// TwinCAT 3 PLC project PLC_OCR
// ProgramVersion: 3.1.4024.0
// libraries:
//   Tc2_Standard, * (Beckhoff Automation GmbH)
//   Tc2_System, * (Beckhoff Automation GmbH)
//   Tc3_Module, * (Beckhoff Automation GmbH)
//   Tc3_Vision, * (Beckhoff Automation GmbH)
// project tree:
//   / PlcTask.TcTTO
//   POUs/ F_GetROI.TcPOU, MAIN.TcPOU
// real-time tasks:
//   TASK PlcTask: cycle T#20ms, priority 20, ADS port 350
//   TASK VnTask ImgAcq (FileSource1): cycle T#10ms, priority 5, ADS port 351

CONFIGURATION PLC_OCR
    RESOURCE PLC ON TwinCAT3
        TASK PlcTask(INTERVAL := T#20ms, PRIORITY := 20);
        PROGRAM MAIN WITH PlcTask : MAIN;
    END_RESOURCE
END_CONFIGURATION

// ---- POUs/MAIN.TcPOU
PROGRAM MAIN
VAR
	bInitialized 		: 	BOOL := FALSE;
	bDeinitialize		:	BOOL;
	bCheck				:	BOOL;
	fbInit 				: 	FB_VN_InitializeFunction;	
	nReturnCode			:   UDINT;
	
	hr					:	HRESULT;
	hrCheck				:	HRESULT;
	hrDeinitialize		:	HRESULT;
	hrOCR				:	HRESULT;
	fbCameraControl		:	FB_VN_FileSourceControl;
	eCameraState		:	ETcVnCameraState;
	sFileName 			: 	STRING;
	ImageCounter		:	UINT;

	stPixelFormat		:	TcVnPixelFormat;
	stRoi				:	TcVnRectangle_UDINT;
	fThreshold			:	LREAL;
	bInvertImage		:	BOOL := TRUE;
	
	ipOriginalImage		:	ITcVnImage; 
	ipBinaryImage		:	ITcVnImage; 
	ipThreshBorder		:	ITcVnImage;
	ipStructElem		: 	ITcvnImage;
	ipOriginImageDisp	:	ITcVnDisplayableImage;
	ipBinImageDisp		:	ITcVnDisplayableImage;
	ipThreshBorderDisp	:	ITcVnDisplayableImage;
	
	aRedColor			: 	TcVnVector4_LREAL := [255,0,0];
	aGreenColor			: 	TcVnVector4_LREAL := [0,255,0];
	aBlueColor			: 	TcVnVector4_LREAL := [0,0,255];
	aWhiteColor			: 	TcVnVector4_LREAL := [255,255,255];
	
	// OCR
	bUseExpFunction		:	BOOL := FALSE;
	ipOCRResult 		:	ITcVnContainer; (* Returns the detected characters (ContainerType_Vector_String_SINT) *)
	sText 				: 	STRING(255);
	nStringLenght		:	INT;

	// OCR Exp
	sPattern			:	STRING;			(* String template containing the format in which characters are presented *)
	eOcrOptions			:	UDINT;			(* Specifies which options must be applied to the function (ETcVnOcrOptions) *)
	ipBoundingBoxes		:	ITcVnContainer;	(* Returns the corresponding bounding boxes of the detected characters (ContainerType_Vector_TcVnRectangle_DINT, optional, set to 0 if not required) *)
	ipConfidences		:	ITcVnContainer;	(* Returns the corresponding classification confidences of the detected characters (ContainerType_Vector_REAL, optional, set to 0 if not required) *)
	fMinConfidence		:	REAL;			(* Returns the minimum value of the confidences *)
	
	nNumberOfElements	: 	ULINT;
	nIterator			: 	ULINT;
	aConfidences		:	ARRAY [0..11] OF REAL;
	stRectangle			:	TcVnRectangle_DINT;
END_VAR

// Disclaimer

// This publication contains statements about the suitability of our products for certain
// areas of application. These statements are based on typical features of our products.
// The examples shown in this publication are for demonstration purposes only.
// The information provided herein should not be regarded as specific operation characteristics.
// It is incumbent on the customer to check and decide whether a product is suitable for use
// in a particular application. We do not give any warranty that the source code which is
// made available with this publication is complete or accurate.

// THE SAMPLE CODE CONTAINED IN THIS PUBLICATION IS PROVIDED “AS IS” WITHOUT WARRANTY OF ANY KIND,
// EITHER EXPRESSED, IMPLIED OR STATUTORY, INCLUDING WITHOUT LIMITATION, ANY WARRANTY WITH RESPECT TO NON-INFRINGEMENT,
// FREEDOM FROM PROPRIETARY RIGHTS OF THIRD PARTIES OR FITNESS FOR ANY PARTICULAR PURPOSE.

// This publication may be changed from time to time without prior notice.
// No liability is assumed for errors and/or omissions.
// Our products are described in detail in our data sheets and documentations.
// Product-specific warnings and cautions must be observed.
// For the latest version of our data sheets and documentations visit our website (www.beckhoff.de).

// © Beckhoff Automation GmbH & Co. KG, December 2023

// The reproduction, distribution and utilization of this document as well as the communication
// of its contents to others without express authorization is prohibited. 
// Offenders will be held liable for the payment of damages.
// All rights reserved in the event of the grant of a patent, utility model or design.

//	==========================================================================================

// SAMPLE - OCR (Optical Character Recognition)
//	-------------------------------------------------------

// Steps To Do:
// ------------
// 1. Add the sample images to the FileSource1 Control
// 2. Activate the Configuration -> Start TwinCAT System and PLC to run -> watch the results in the ADS Image Watch
// 3. Switch between OCR standard and expert function with bUseExpFunction

// Load OCR Model
IF NOT bInitialized THEN
	fbInit(eFunction := TCVN_IF_OCR, nOptions := ETcVnOcrModelType.TCVN_OMT_NUMBERS_SC_UCLETTERS OR ETcVnOcrModelType.TCVN_OMT_NUMBERS_SC OR ETcVnOcrModelType.TCVN_OMT_UCLETTERS, bStart := TRUE);
	
	IF NOT fbInit.bBusy THEN
		fbInit(bStart := FALSE);
		IF NOT fbInit.bError THEN
			bInitialized := TRUE;
			nReturnCode := fbInit.nErrorId AND 16#FFF;
		ELSE
			nReturnCode := fbInit.nErrorId AND 16#FFF;
		END_IF
	END_IF
END_IF

// Check if Model is initialized
IF bCheck THEN
	bCheck := FALSE;
	hrCheck := F_VN_CheckFunctionInitialization(eFunction := TCVN_IF_OCR, nOptions := ETcVnOcrModelType.TCVN_OMT_NUMBERS_SC, hrPrev := S_OK);
END_IF

// Unload OCR Model
IF bDeinitialize THEN
	bDeinitialize := FALSE;
	hrDeinitialize := F_VN_DeinitializeFunction(eFunction:= TCVN_IF_OCR, nOptions:= ETcVnOcrModelType.TCVN_OMT_NUMBERS_SC, hrPrev:= S_OK);
	bInitialized := FALSE;
END_IF

// Get Camera State
eCameraState := fbCameraControl.GetState();
	
// CameraControl is in error state, so try to reset the camera connection
IF eCameraState = TCVN_CS_ERROR THEN
	hr := fbCameraControl.Reset();

// Camera not yet streaming
ELSIF eCameraState < TCVN_CS_ACQUIRING THEN
	hr := fbCameraControl.StartAcquisition();

// Camera streaming
ELSIF eCameraState = TCVN_CS_ACQUIRING THEN	
	
	hr := fbCameraControl.GetCurrentImageAndFileName(ipImage := ipOriginalImage, sFileName := sFileName, 80);
	
	IF bInitialized AND SUCCEEDED(hr) AND ipOriginalImage <> 0 THEN
		
		ImageCounter := ImageCounter + 1;
		
		// Check pixel format and prepare work image
		hr := F_VN_GetPixelFormat(ipOriginalImage, stPixelFormat, hr);			
		IF stPixelFormat.nChannels = 3 AND stPixelFormat.ePixelEncoding = TCVN_PE_NONE THEN
			hr := F_VN_ConvertColorSpace(ipOriginalImage, ipBinaryImage, TCVN_CST_RGB_TO_GRAY, hr);			
		ELSE
			hr := F_VN_CopyImage(ipOriginalImage, ipBinaryImage, hr);
		END_IF
		
		// Helper funtion to get ROI and threshold value according to sample image
		F_GetROI(sFileName, stRoi, fThreshold, bInvertImage, sPattern);
			 
		// Set ROI and draw rectangle
		hr := F_VN_SetRoi_TcVnRectangle_UDINT(stRoi, ipBinaryImage, hr);
		hr := F_VN_DrawRectangle_TcVnRectangle_UDINT(stRoi, ipOriginalImage, aRedColor, 2, hr);
		
		// Filter Image 
		// Add or replace pre-processing functions if needed
		hr := F_VN_CreateStructuringElement(ipStructElem, ETcVnStructuringElementShape.TCVN_SES_RECTANGLE, 3,3, hr);
		hr := F_VN_MorphologicalOperator(ipBinaryImage, ipBinaryImage, ETcvnMorphologicalOperator.TCVN_MO_OPENING, ipStructElem, hr);	
		
		// Invert image depending on bright or dark text color 
		IF bInvertImage THEN
			hr := F_VN_Threshold(ipBinaryImage, ipBinaryImage, fThreshold, 255, TCVN_TT_BINARY_INV, hr);
		ELSE
			hr := F_VN_Threshold(ipBinaryImage, ipBinaryImage, fThreshold, 255, TCVN_TT_BINARY, hr);
		END_IF
		
		// Remove border objects
		hr := F_VN_BrightBorderObjects(ipBinaryImage, ipThreshBorder, hr);
		hr := F_VN_SubtractImages(ipBinaryImage, ipThreshBorder, ipBinaryImage, hr);
	
		// Read characters
		IF NOT bUseExpFunction THEN
			hrOCR := F_VN_OCR(
					ipSrcImage		:= ipBinaryImage,
					eModel			:= ETcVnOcrModelType.TCVN_OMT_NUMBERS_SC_UCLETTERS,
					ipCharacters	:= ipOCRResult,
					hrPrev			:= hr);
		ELSE
			hrOCR := F_VN_OCRExp(
					ipSrcImage		:= ipBinaryImage,
					eModel			:= ETcVnOcrModelType.TCVN_OMT_NUMBERS_SC or ETcVnOcrModelType.TCVN_OMT_UCLETTERS,
					ipCharacters	:= ipOCRResult, 
					sPattern		:= sPattern,
					eOcrOptions		:= eOcrOptions,
					ipBoundingBoxes	:= ipBoundingBoxes, 
					ipConfidences	:= ipConfidences,
					hrPrev			:= hr,
					fMinConfidence	=> fMinConfidence);
		END_IF
				
		// Check if characters were found
		hr := F_VN_GetNumberOfElements(ipOCRResult, nNumberOfElements, hrOCR);
		IF SUCCEEDED(hr) AND nNumberOfElements > 0 THEN
			// Export character to string
			hr := F_VN_ExportSubContainer_String(ipOCRResult, 0, sText, 255, hr);
			nStringLenght := LEN(sText);
			
			// Write text result to filtered and original image
			hr := F_VN_PutText(sText, ipBinaryImage, 12, 12, TCVN_FT_HERSHEY_PLAIN, 1, aWhiteColor, hr);
			hr := F_VN_PutText(sText, ipOriginalImage, stRoi.nX + 5, stRoi.nY + 25, TCVN_FT_HERSHEY_DUPLEX, 1, aGreenColor, hr);
			
			IF bUseExpFunction THEN 
				// Get number of Confidence elements and export them if array is large enough 
				MEMSET(ADR(aConfidences), 0, SIZEOF(aConfidences));
				hr := F_VN_GetNumberOfElements(ipConfidences, nNumberOfElements, hr);
				
				// Check if number of elements fits to array size
				IF nNumberOfElements > 0 AND nNumberOfElements <= 12 THEN
					hr := F_VN_ExportContainer(ipConfidences, ADR(aConfidences), SIZEOF(aConfidences), hr);
				END_IF
				
				// Get bounding box rectangle and draw it to filtered and original image
				hr := F_VN_GetNumberOfElements(ipBoundingBoxes, nNumberOfElements, hr);
				IF nNumberOfElements > 0 THEN
					FOR nIterator := 0 TO nNumberOfElements -1 DO
						hr := F_VN_GetAt_TcVnRectangle_DINT(ipBoundingBoxes, stRectangle, nIterator, hr);
						hr := F_VN_DrawRectangle_TcVnRectangle_DINT(stRectangle, ipBinaryImage, aWhiteColor, 1, hr);
						// Add ROI Offset
						stRectangle.nX := stRectangle.nX + UDINT_TO_DINT(stRoi.nX);
						stRectangle.nY := stRectangle.nY + UDINT_TO_DINT(stRoi.nY);
						hr := F_VN_DrawRectangle_TcVnRectangle_DINT(stRectangle, ipOriginalImage, aBlueColor, 1, hr);
					END_FOR
				END_IF
			END_IF
		END_IF
		
		// Display images
		hr := F_VN_TransformIntoDisplayableImage(ipOriginalImage, ipOriginImageDisp, S_OK);
		hr := F_VN_TransformIntoDisplayableImage(ipBinaryImage, ipBinImageDisp, S_OK);
		hr := F_VN_TransformIntoDisplayableImage(ipThreshBorder, ipThreshBorderDisp, S_OK);
		
		// Release Pointer
		hr := FW_SafeRelease(ADR(ipOCRResult));
		hr := FW_SafeRelease(ADR(ipBoundingBoxes));
		hr := FW_SafeRelease(ADR(ipConfidences));
	END_IF
END_IF

END_PROGRAM

// ---- POUs/F_GetROI.TcPOU
FUNCTION F_GetROI : HRESULT
VAR_INPUT
	sFileName 			: 	REFERENCE TO STRING;
	stRoi				:	REFERENCE TO TcVnRectangle_UDINT;
	fThreshold			:	REFERENCE TO LREAL;
	bInvertImage		: 	REFERENCE TO BOOL;
	sPattern			:	REFERENCE TO STRING;
END_VAR
VAR
END_VAR

IF sFileName = 'OCR_01.png' THEN
	stRoi.nX := 86;
	stRoi.nY := 34;
	stRoi.nWidth := 263;
	stRoi.nHeight := 102;
	fThreshold := 150;
	bInvertImage := TRUE;
	sPattern := 'dd#dd#dd';
ELSIF sFileName = 'OCR_02.png' THEN
	stRoi.nX := 69;
	stRoi.nY := 40;
	stRoi.nWidth := 237;
	stRoi.nHeight := 80;
	fThreshold := 150;
	bInvertImage := TRUE;
	sPattern := 'dd#dd#dddd';
ELSIF sFileName = 'OCR_03.png' THEN
	stRoi.nX := 30;
	stRoi.nY := 40;
	stRoi.nWidth := 460;
	stRoi.nHeight := 110;
	fThreshold := 120;
	bInvertImage := TRUE;
	sPattern := 'udddudd###d';
ELSIF sFileName = 'OCR_04.png' THEN
	stRoi.nX := 131;
	stRoi.nY := 25;
	stRoi.nWidth := 243;
	stRoi.nHeight := 83;
	fThreshold := 75;
	bInvertImage := TRUE;
	sPattern := 'dd#dd#dddd';
ELSIF sFileName = 'OCR_05.png' THEN
	stRoi.nX := 129;
	stRoi.nY := 78;
	stRoi.nWidth := 257;
	stRoi.nHeight := 115;
	fThreshold := 150;
	bInvertImage := TRUE;
	sPattern := 'dd#dd#dd';
ELSIF sFileName = 'OCR_06.png' THEN
	stRoi.nX := 71;
	stRoi.nY := 50;
	stRoi.nWidth := 293;
	stRoi.nHeight := 101;
	fThreshold := 75;
	bInvertImage := TRUE;
	sPattern := 'dd#dd#dddd';
ELSIF sFileName = 'OCR_07.png' THEN
	stRoi.nX := 50;
	stRoi.nY := 120;
	stRoi.nWidth := 470;
	stRoi.nHeight := 110;
	fThreshold := 140;
	bInvertImage := FALSE;
	sPattern := 'udddudd###';
ELSIF sFileName = 'OCR_08.png' THEN
	stRoi.nX := 100;
	stRoi.nY := 83;
	stRoi.nWidth := 276;
	stRoi.nHeight := 108;
	fThreshold := 165;
	bInvertImage := TRUE;
	sPattern := 'dd#dd#dd';
ELSIF sFileName = 'OCR_09.png' THEN
	stRoi.nX := 90;
	stRoi.nY := 103;
	stRoi.nWidth := 284;
	stRoi.nHeight := 82; 
	fThreshold := 178;
	bInvertImage := TRUE;
	sPattern := 'dd#dd#dddd';
ELSIF sFileName = 'OCR_10.png' THEN
	stRoi.nX := 207;
	stRoi.nY := 4;
	stRoi.nWidth := 283;
	stRoi.nHeight := 104;
	fThreshold := 130;
	bInvertImage := TRUE;
	sPattern := 'dd#dd#dddd';
ELSIF sFileName = 'OCR_11.png' THEN
	stRoi.nX := 175;
	stRoi.nY := 245;
	stRoi.nWidth := 660;
	stRoi.nHeight := 115;
	fThreshold := 160;
	bInvertImage := TRUE;
	sPattern := 'uu#dddddddd';	
ELSIF sFileName = 'OCR_12.png' THEN 
	stRoi.nX := 74;
	stRoi.nY := 198;
	stRoi.nWidth := 248;
	stRoi.nHeight := 95;
	fThreshold := 130;
	bInvertImage := FALSE;
	sPattern := 'dd#dddd';
ELSIF sFileName = 'OCR_13.png' THEN
	stRoi.nX := 404;
	stRoi.nY := 2;
	stRoi.nWidth := 392;
	stRoi.nHeight := 159;
	fThreshold := 130;
	bInvertImage := FALSE;
	sPattern := 'dd#dd#dd';
ELSIF sFileName = 'OCR_14.png' THEN
	stRoi.nX := 260;
	stRoi.nY := 105;
	stRoi.nWidth := 340;
	stRoi.nHeight := 102;
	fThreshold := 160;
	bInvertImage := FALSE;
	sPattern := 'dd#dd#dddd';
ELSIF sFileName = 'OCR_15.png' THEN
	stRoi.nX := 250;
	stRoi.nY := 5;
	stRoi.nWidth := 560;
	stRoi.nHeight := 125;
	fThreshold := 160;
	bInvertImage := TRUE;
	sPattern := 'uddddd#dd#dd';
ELSIF sFileName = 'OCR_16.png' THEN
	stRoi.nX := 200;
	stRoi.nY := 0;
	stRoi.nWidth := 285;
	stRoi.nHeight := 70;
	fThreshold := 130;
	bInvertImage := FALSE;
	sPattern := 'dd#dd#dddd';
ELSIF sFileName = 'OCR_17.png' THEN
	stRoi.nX := 247;
	stRoi.nY := 83;
	stRoi.nWidth := 213;
	stRoi.nHeight := 94;
	fThreshold := 155;
	bInvertImage := FALSE;
	sPattern := 'dd#dddd';
ELSIF sFileName = 'OCR_18.png' THEN
	stRoi.nX := 25;
	stRoi.nY := 187;
	stRoi.nWidth := 330;
	stRoi.nHeight := 109;
	fThreshold := 100;
	bInvertImage := FALSE;
	sPattern := 'dd#dddd';
ELSIF sFileName = 'OCR_19.png' THEN
	stRoi.nX := 365;
	stRoi.nY := 70;
	stRoi.nWidth := 300;
	stRoi.nHeight := 95;
	fThreshold := 80;
	bInvertImage := TRUE;
	sPattern := 'uduuuud';
END_IF

END_FUNCTION
